// TIA Portal V16 export
// export: Created 2024-12-03T15:41:40.0441336Z, ExportSetting WithDefaults, DisplayName Totally Integrated Automation Portal, DisplayVersion V16 Update 6, DisplayName TIA Portal Version Control Interface, DisplayVersion V16 Update 2, DisplayName TIA Portal Openness, DisplayVersion V16 Update 6, DisplayName TIA Portal Teamcenter Gateway, DisplayVersion V16, DisplayName SINAMICS Startdrive Advanced, DisplayVersion V16 Update 5, DisplayName SINAMICS Startdrive G130, G150, S120, S150, SINAMICS MV, S210, DisplayVersion V16 Update 5, DisplayName SINAMICS Startdrive G110M, G120, G120C, G120D, G120P, G115D, DisplayVersion V16 Update 5, DisplayName STEP 7 Professional, DisplayVersion V16 Update 6, DisplayName STEP 7 Safety, DisplayVersion V16, DisplayName WinCC Advanced / Unified PC, DisplayVersion V16 Update 6
FUNCTION_BLOCK "DRV_CONTROLLER_FB"   // FB3, SCL
{ S7_Optimized_Access := 'TRUE' }
VERSION : 0.1
// stored: AutoNumber true, IsIECCheckEnabled false, IsRetainMemResEnabled false, MemoryReserve 100, SetENOAutomatically false, UDAEnableTagReadback false
   VAR
      DRV_101_DRV_1 : "Nord_DriveController";
   END_VAR
BEGIN
   REGION DRV_101_DRV_1

       "Conv_Nord_Drive_Commander"(I_Conv := "CONV_DB".CONV_101,
                                   I_INV := FALSE,
                                   IO_NordDrive := "DRV_DB".DRV_101_DRV_1);

       #DRV_101_DRV_1(I_MotorData := "I_DRV_101_1",
                      I_Interlock := FALSE,
                      I_TimeNotRunning := T#10s,
                      I_TimeNotStopping := T#10s,
                      I_SlowStopMode := FALSE,
                      IO_MotorData := "Q_DRV_101_1",
                      IO_MotorStatus := "DRV_DB".DRV_101_DRV_1);

   END_REGION
END_FUNCTION_BLOCK
